// TIA Portal V20 export
// export: Created 2025-12-01T14:57:23.4142356Z, ExportSetting None, DisplayName Totally Integrated Automation Portal, DisplayVersion V20 Update 3, DisplayName TIA Portal Openness, DisplayVersion V20 Update 3, DisplayName TIA Portal Version Control Interface, DisplayVersion V20 Update 3, DisplayName STEP 7 Professional, DisplayVersion V20 Update 3, DisplayName STEP 7 Safety, DisplayVersion V20 Update 2, DisplayName WinCC Basic/Comfort/Advanced, DisplayVersion V20 Update 3, DisplayName WinCC Professional, DisplayVersion V20 Update 3, DisplayName WinCC Unified, DisplayVersion V20 Update 3
DATA_BLOCK "DB910_Conf_Sistema_Transporte"   // DB910
{ S7_Optimized_Access := 'FALSE' }
AUTHOR : GENERAL
NAME : 20130301
VERSION : 3.0
// stored: AutoNumber false
   VAR RETAIN
      TiemposTracking : Struct
         V_CNT_pHsMx_E1E3 : Int := 300;
         V_CNT_pHsMx_FTF_E1E3 : Int := 200;
         V_CNTSeg_pHsMX_E1E3 : Int := 2000;
         V_CNT_Paso_Lenta_E1E3 : Int := 1000;
         V_CNT_pHsMx_E2E4 : Int := 400;
         V_CNT_pHsMx_FTF_E2E4 : Int := 200;
         V_CNTSeg_pHsMX_E2E4 : Int := 1000;
         V_CNT_Paso_Lenta_E2E4 : Int := 1000;
         V_CNT_ApHsMx : Int := 100;
         V_CNTSeg_ApHsMx : Int := 2000;
         V_Subir_TP_Min : Int := 1000;
         V_Bajar_TP_Max : Int := 3000;
         V_CNT_Separacion : Int := 1000;
         V_CNT_SubirTPCentral : Int := 2500;
         V_CNT_Simultaneo : Int := 100;
         V_InicioSimultaneo : Int := 0;
         V_FinalSimultaneo : Int := 0;
         V_TIM_BLOQUEO : Int := 4500;
         V_PasoLenta_0 : Int := 2500;
         V_PasoLenta_90 : Int := 2500;
         Ret_Paso_Lenta_Var : Int := 6;
         V_TMP_Retirar : Int := 5000;
         V_CNT_Centrado : Int := 2000;
         V_CNT_Reposo : Int := 3000;
      END_STRUCT;
      TiemposTOut : Struct
         V_TOut_Tx_Mx_E1 : Int := 7;   // En Segundos
         V_TOut_Tx_Mx_E2 : Int := 7;   // En Segundos
         V_TOut_TP : Int := 2000;   // En milisegundos
         V_TOut_TR : Int := 2000;   // En milisegundos
         V_TOut_MAQ : Int := 2000;   // En milisegundos
         V_TOut_Elev : Int := 2000;   // En milisegundos
         V_TOut_MElev : Int := 10000;   // En milisegundos
         V_TOut_MG : Int := 10000;   // En milisegundos
         V_TOut_Interlock : Int := 10000;   // En milisegundos
         V_TMP_Protrusion : Int := 200;   // En milisegundos
         V_PerdidapHs : Int := 500;   // En milisegundos
      END_STRUCT;
      TiemposRouting : Struct
         V_Paro : DInt := 3000;
         V_CNT_ApHsMx_E1 : DInt := 200;
         V_CNT_ApHsMx_E2 : DInt := 200;
         V_CNT_ApHsMx_E3 : DInt := 200;
         V_CNT_ApHsMx_E4 : DInt := 200;
         V_CNT_ApHsMx_S1 : DInt := 200;
         V_CNT_ApHsMx_S2 : DInt := 200;
         V_CNT_ApHsMx_S3 : DInt := 200;
         V_CNT_ApHsMx_S4 : DInt := 200;
         V_Vaciado : DInt := 10000;
         V_Gap : DInt := 200;
      END_STRUCT;
      TiemposTOutRouting : Struct
         V_TOut_Tx_Mx_E1 : DInt := 5000;
         V_TOut_Tx_Mx_E2 : DInt := 5000;
         V_TOut_TP : DInt := 2000;
         V_TOut_TR : DInt := 2000;
         V_TOut_MAQ : DInt := 2000;
         V_TOut_Elev : DInt := 2000;
         V_TMP_Protrusion : DInt := 200;
         V_TOut_Empujador : DInt := 3000;
      END_STRUCT;
      Tiempo_Decel_SM_E1S3 : Int;
      Tiempo_Decel_SM_E2S4 : Int;
      Tiempo_Decel_SM_ELEV : Int;
   END_VAR
BEGIN
END_DATA_BLOCK
